TYPE TModuleCommands :
	(
		MC_NoCmd,
		MC_Init,
		MC_Manual,
		MC_Stop,
		MC_Run
	);
END_TYPE

(* stored: Version 1.1.0.1, ProductVersion 3.1.4022.12
   DUT TModuleCommands: Id {652ca473-2db9-44d5-89b7-a46dbd6fb350} *)
